INTERFACE I_Instance EXTENDS __SYSTEM.IQueryInterface

PROPERTY PUBLIC NameSpace : STRING
GET
END_GET
END_PROPERTY

METHOD PUBLIC SharesNamespaceWith : BOOL
VAR_INPUT
	OtherInstance : I_Instance;
END_VAR
END_METHOD

END_INTERFACE

(* stored: Version 1.1.0.1, ProductVersion 3.1.4024.11
   Itf I_Instance: Id {e9c4db03-2c6d-45c9-bf2c-c529468a9350}
   Property NameSpace: Id {06ec18fe-fdbc-4508-8f50-422b00a4c140}
   Get Get: Id {ce4836ba-28a1-4dfe-977b-31699c1034c1}
   Method SharesNamespaceWith: Id {ff664b26-639f-43da-a6be-9181b0924d9b} *)
